// TIA Portal V17 export
// export: Created 2024-06-19T09:47:14.9665731Z, ExportSetting WithDefaults, DisplayName Totally Integrated Automation Portal, DisplayVersion V17, DisplayName TIA Portal Openness, DisplayVersion V17, DisplayName TIA Portal Version Control Interface, DisplayVersion V17, DisplayName STEP 7 Professional, DisplayVersion V17, DisplayName STEP 7 Safety, DisplayVersion V17, DisplayName WinCC Professional, DisplayVersion V17
VAR_GLOBAL   // PLC tag table "St1_Out"
   IO_Ouverture_Pinces AT %Q1.2 : Bool;   // Ouverture : Pinces de préhension
   IO_Fermeture_Pinces AT %Q1.3 : Bool;   // Fermeture : Pinces de préhension
   IO_Vy_PileAV AT %Q1.4 : Bool;   // Conditions sur voyant C2 : OK
   IO_Vy_PileAR AT %Q1.5 : Bool;   // Conditions sur voyant C4 : OK
END_VAR
